// TIA Portal V18 export
FUNCTION "07_Speed Control" : Void   // FC8, F_LAD
TITLE = Manage Safety Encoder
{ S7_Optimized_Access := 'TRUE' }
BEGIN
END_FUNCTION
